# EPICS substitutions: iocs/es3602-test/es3602testApp/Db/es3602-test.substitutions
file es3602-channel.db
{

}
